(* IEC 61131-3 sources: RL_MAR/experiments/comparison/autoplc/results/gpt-4o_20260511_211137/med_44, 1 file *)

(* ---- med_44_1.st ---- *)
FUNCTION_BLOCK DroneChargingStation
VAR_INPUT
    Drone1BatteryLevel : INT := 0; (* Battery level of Drone 1 (0-100%) *)
    Drone2BatteryLevel : INT := 0; (* Battery level of Drone 2 (0-100%) *)
    Drone3BatteryLevel : INT := 0; (* Battery level of Drone 3 (0-100%) *)
    ChargingTime : TIME := T#30s; (* Charging time required for each drone *)
END_VAR
VAR_OUTPUT
    Drone1Status : BOOL := FALSE; (* Status of Drone 1 *)
    Drone2Status : BOOL := FALSE; (* Status of Drone 2 *)
    Drone3Status : BOOL := FALSE; (* Status of Drone 3 *)
    ChargingStationStatus : BOOL := FALSE; (* Charging station status *)
    DroneDeployed : BOOL := FALSE; (* Indicates if a drone is deployed *)
END_VAR
VAR
    TimeRemaining : TIME := T#0s; (* Remaining charging time for the current charging operation *)
END_VAR

(* Initialization *)
IF NOT ChargingStationStatus THEN
    Drone1Status := FALSE;
    Drone2Status := FALSE;
    Drone3Status := FALSE;
    DroneDeployed := FALSE;
    TimeRemaining := ChargingTime;
END_IF

(* Idle State Logic *)
IF NOT ChargingStationStatus THEN
    IF Drone1BatteryLevel < 20 THEN
        Drone1Status := TRUE;
        ChargingStationStatus := TRUE;
    ELSIF Drone2BatteryLevel < 20 THEN
        Drone2Status := TRUE;
        ChargingStationStatus := TRUE;
    ELSIF Drone3BatteryLevel < 20 THEN
        Drone3Status := TRUE;
        ChargingStationStatus := TRUE;
    END_IF
END_IF

(* Charging State Logic *)
IF ChargingStationStatus THEN
    IF TimeRemaining > T#0s THEN
        TimeRemaining := TimeRemaining - T#1s; (* Decrement time by 1 second *)
    ELSE
        Drone1Status := FALSE;
        Drone2Status := FALSE;
        Drone3Status := FALSE;
        ChargingStationStatus := FALSE;
        TimeRemaining := ChargingTime; (* Reset for next cycle *)
    END_IF
END_IF

(* Deployment State Logic *)
IF DroneDeployed THEN
    IF Drone1BatteryLevel < 10 OR Drone2BatteryLevel < 10 OR Drone3BatteryLevel < 10 THEN
        DroneDeployed := FALSE; (* Recall the drone *)
    END_IF
END_IF

END_FUNCTION_BLOCK
